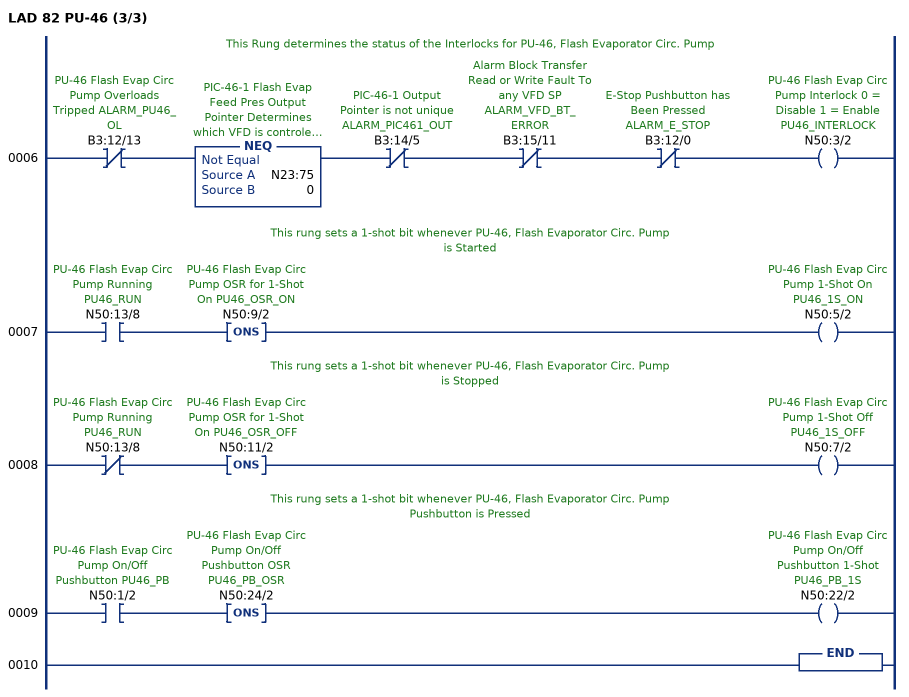
% Rung: 6 %
% This Rung determines the status of the Interlocks for PU-46, Flash Evaporator Circ. Pump %
SOR XIO B3:12/13 NEQ N23:75 0 XIO B3:14/5 XIO B3:15/11 XIO B3:12/0 OTE N50:3/2 EOR
%   B3:12/13  ALARM_PU46_OL  "PU-46 Flash Evap Circ Pump Overloads Tripped" %
%   N23:75  PIC461_OUT_PTR  "PIC-46-1 Flash Evap Feed Pres Output Pointer Determines which VFD is controled by FIC" %
%   B3:14/5  ALARM_PIC461_OUT  "PIC-46-1 Output Pointer is not unique" %
%   B3:15/11  ALARM_VFD_BT_ERROR  "Alarm Block Transfer Read or Write Fault To any VFD SP" %
%   B3:12/0  ALARM_E_STOP  "E-Stop Pushbutton has Been Pressed" %
%   N50:3/2  PU46_INTERLOCK  "PU-46 Flash Evap Circ Pump Interlock 0 = Disable 1 = Enable" %
% Rung: 7 %
% This rung sets a 1-shot bit whenever PU-46, Flash Evaporator Circ. Pump
% is Started %
SOR XIC N50:13/8 OSR N50:9/2 OTE N50:5/2 EOR
%   N50:13/8  PU46_RUN  "PU-46 Flash Evap Circ Pump Running" %
%   N50:9/2  PU46_OSR_ON  "PU-46 Flash Evap Circ Pump OSR for 1-Shot On" %
%   N50:5/2  PU46_1S_ON  "PU-46 Flash Evap Circ Pump 1-Shot On" %
% Rung: 8 %
% This rung sets a 1-shot bit whenever PU-46, Flash Evaporator Circ. Pump
% is Stopped %
SOR XIO N50:13/8 OSR N50:11/2 OTE N50:7/2 EOR
%   N50:13/8  PU46_RUN  "PU-46 Flash Evap Circ Pump Running" %
%   N50:11/2  PU46_OSR_OFF  "PU-46 Flash Evap Circ Pump OSR for 1-Shot On" %
%   N50:7/2  PU46_1S_OFF  "PU-46 Flash Evap Circ Pump 1-Shot Off" %
% Rung: 9 %
% This rung sets a 1-shot bit whenever PU-46, Flash Evaporator Circ. Pump
% Pushbutton is Pressed %
SOR XIC N50:1/2 OSR N50:24/2 OTE N50:22/2 EOR
%   N50:1/2  PU46_PB  "PU-46 Flash Evap Circ Pump On/Off Pushbutton" %
%   N50:24/2  PU46_PB_OSR  "PU-46 Flash Evap Circ Pump On/Off Pushbutton OSR" %
%   N50:22/2  PU46_PB_1S  "PU-46 Flash Evap Circ Pump On/Off Pushbutton 1-Shot" %
% Rung: 10 %
SOR END EOR

LADDER 86 "ALL VFDS"    % Control All VFD's %
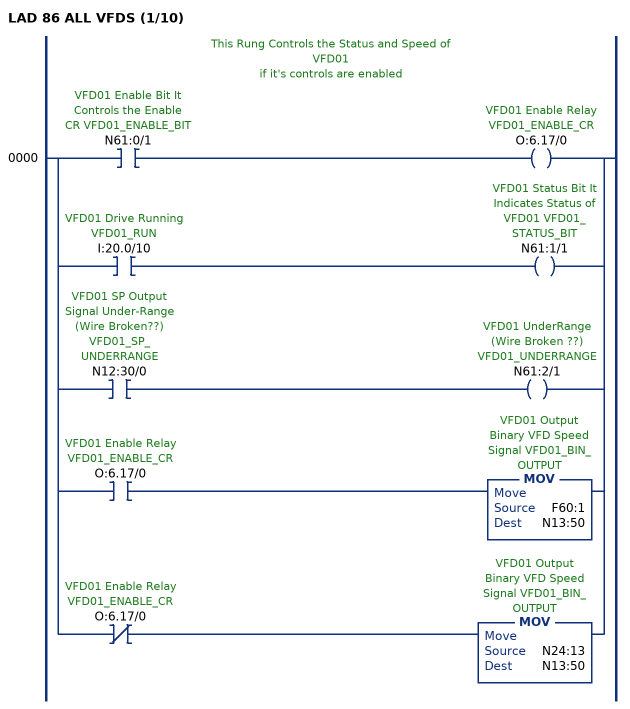
% Rung: 0 %
% This Rung Controls the Status and Speed of
% VFD01
% if it's controls are enabled %
SOR BST XIC N61:0/1 OTE O:6.17/0 NXB XIC I:20.0/10 OTE N61:1/1 NXB XIC N12:30/0 OTE N61:2/1 NXB XIC O:6.17/0 MOV F60:1 N13:50 NXB XIO O:6.17/0 MOV N24:13 N13:50 BND EOR
%   N61:0/1  VFD01_ENABLE_BIT  "VFD01 Enable Bit It Controls the Enable CR" %
%   O:6.17/0  VFD01_ENABLE_CR  "VFD01 Enable Relay" %
%   I:20.0/10  VFD01_RUN  "VFD01 Drive Running" %
%   N61:1/1  VFD01_STATUS_BIT  "VFD01 Status Bit It Indicates Status of VFD01" %
%   N12:30/0  VFD01_SP_UNDERRANGE  "VFD01 SP Output Signal Under-Range (Wire Broken??)" %
%   N61:2/1  VFD01_UNDERRANGE  "VFD01 UnderRange (Wire Broken ??)" %
%   F60:1  VFD01_BIN  "VFD01 VFD Table Value (is sent to Actual AO Location for VFD)" %
%   N13:50  VFD01_BIN_OUTPUT  "VFD01 Output Binary VFD Speed Signal" %
%   N24:13  AO_MIN_OE4  "Analog Output Minimum Value Generates 4 mA DC (To OE4 AO Module)" %

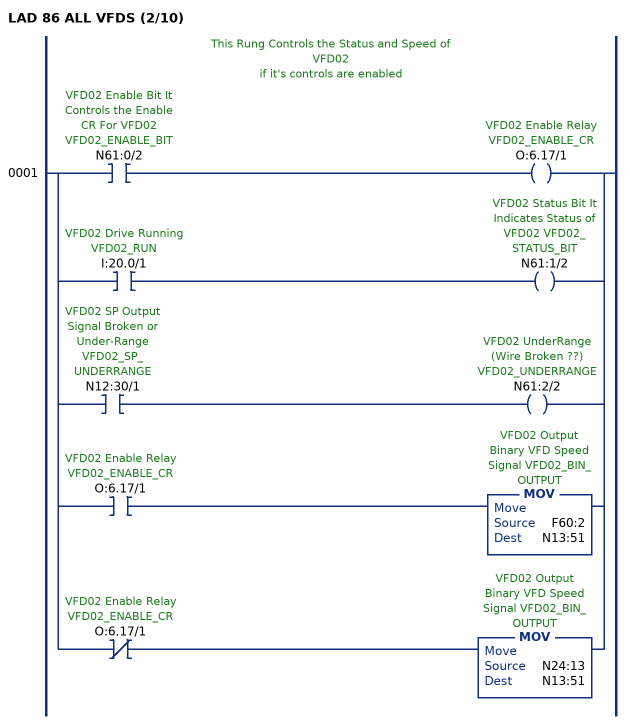
% Rung: 1 %
% This Rung Controls the Status and Speed of
% VFD02
% if it's controls are enabled %
SOR BST XIC N61:0/2 OTE O:6.17/1 NXB XIC I:20.0/1 OTE N61:1/2 NXB XIC N12:30/1 OTE N61:2/2 NXB XIC O:6.17/1 MOV F60:2 N13:51 NXB XIO O:6.17/1 MOV N24:13 N13:51 BND EOR
%   N61:0/2  VFD02_ENABLE_BIT  "VFD02 Enable Bit It Controls the Enable CR For VFD02" %
%   O:6.17/1  VFD02_ENABLE_CR  "VFD02 Enable Relay" %
%   I:20.0/1  VFD02_RUN  "VFD02 Drive Running" %
%   N61:1/2  VFD02_STATUS_BIT  "VFD02 Status Bit It Indicates Status of VFD02" %
%   N12:30/1  VFD02_SP_UNDERRANGE  "VFD02 SP Output Signal Broken or Under-Range" %
%   N61:2/2  VFD02_UNDERRANGE  "VFD02 UnderRange (Wire Broken ??)" %
%   F60:2  VFD02_BIN  "VFD02 VFD Table Value (is sent to Actual AO Location for VFD)" %
%   N13:51  VFD02_BIN_OUTPUT  "VFD02 Output Binary VFD Speed Signal" %
%   N24:13  AO_MIN_OE4  "Analog Output Minimum Value Generates 4 mA DC (To OE4 AO Module)" %

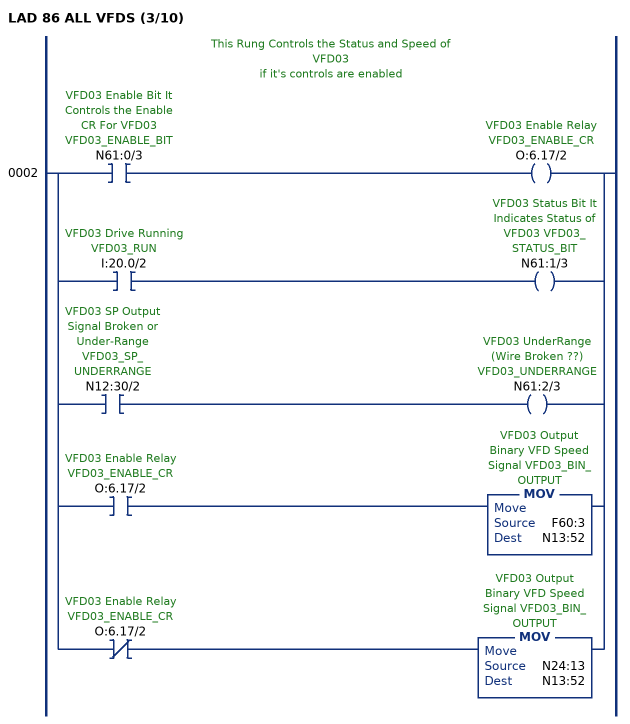
% Rung: 2 %
% This Rung Controls the Status and Speed of
% VFD03
% if it's controls are enabled %
SOR BST XIC N61:0/3 OTE O:6.17/2 NXB XIC I:20.0/2 OTE N61:1/3 NXB XIC N12:30/2 OTE N61:2/3 NXB XIC O:6.17/2 MOV F60:3 N13:52 NXB XIO O:6.17/2 MOV N24:13 N13:52 BND EOR
%   N61:0/3  VFD03_ENABLE_BIT  "VFD03 Enable Bit It Controls the Enable CR For VFD03" %
%   O:6.17/2  VFD03_ENABLE_CR  "VFD03 Enable Relay" %
%   I:20.0/2  VFD03_RUN  "VFD03 Drive Running" %
%   N61:1/3  VFD03_STATUS_BIT  "VFD03 Status Bit It Indicates Status of VFD03" %
%   N12:30/2  VFD03_SP_UNDERRANGE  "VFD03 SP Output Signal Broken or Under-Range" %
%   N61:2/3  VFD03_UNDERRANGE  "VFD03 UnderRange (Wire Broken ??)" %
%   F60:3  VFD03_BIN  "VFD03 VFD Table Value (is sent to Actual AO Location for VFD)" %
%   N13:52  VFD03_BIN_OUTPUT  "VFD03 Output Binary VFD Speed Signal" %
%   N24:13  AO_MIN_OE4  "Analog Output Minimum Value Generates 4 mA DC (To OE4 AO Module)" %

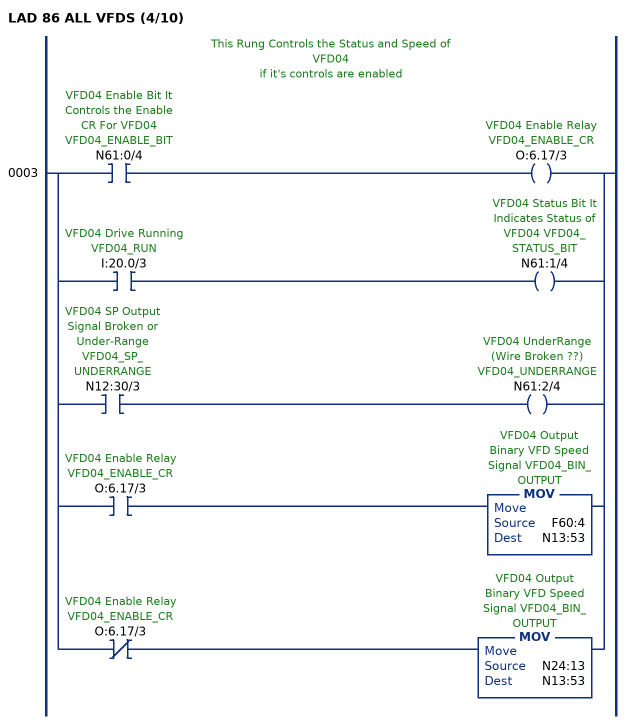
% Rung: 3 %
% This Rung Controls the Status and Speed of
% VFD04
% if it's controls are enabled %
SOR BST XIC N61:0/4 OTE O:6.17/3 NXB XIC I:20.0/3 OTE N61:1/4 NXB XIC N12:30/3 OTE N61:2/4 NXB XIC O:6.17/3 MOV F60:4 N13:53 NXB XIO O:6.17/3 MOV N24:13 N13:53 BND EOR
%   N61:0/4  VFD04_ENABLE_BIT  "VFD04 Enable Bit It Controls the Enable CR For VFD04" %
%   O:6.17/3  VFD04_ENABLE_CR  "VFD04 Enable Relay" %
%   I:20.0/3  VFD04_RUN  "VFD04 Drive Running" %
%   N61:1/4  VFD04_STATUS_BIT  "VFD04 Status Bit It Indicates Status of VFD04" %
%   N12:30/3  VFD04_SP_UNDERRANGE  "VFD04 SP Output Signal Broken or Under-Range" %
%   N61:2/4  VFD04_UNDERRANGE  "VFD04 UnderRange (Wire Broken ??)" %
%   F60:4  VFD04_BIN  "VFD04 VFD Table Value (is sent to Actual AO Location for VFD)" %
%   N13:53  VFD04_BIN_OUTPUT  "VFD04 Output Binary VFD Speed Signal" %
%   N24:13  AO_MIN_OE4  "Analog Output Minimum Value Generates 4 mA DC (To OE4 AO Module)" %

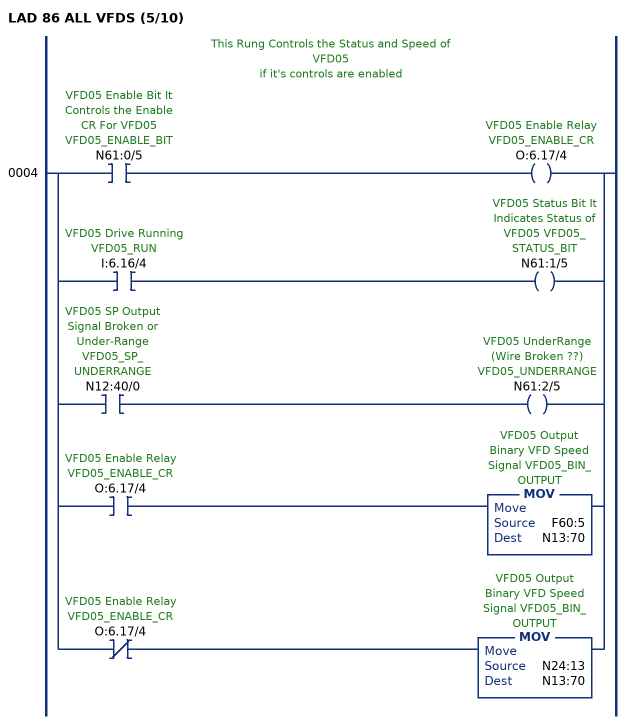
% Rung: 4 %
% This Rung Controls the Status and Speed of
% VFD05
% if it's controls are enabled %
SOR BST XIC N61:0/5 OTE O:6.17/4 NXB XIC I:6.16/4 OTE N61:1/5 NXB XIC N12:40/0 OTE N61:2/5 NXB XIC O:6.17/4 MOV F60:5 N13:70 NXB XIO O:6.17/4 MOV N24:13 N13:70 BND EOR
%   N61:0/5  VFD05_ENABLE_BIT  "VFD05 Enable Bit It Controls the Enable CR For VFD05" %
%   O:6.17/4  VFD05_ENABLE_CR  "VFD05 Enable Relay" %
%   I:6.16/4  VFD05_RUN  "VFD05 Drive Running" %
%   N61:1/5  VFD05_STATUS_BIT  "VFD05 Status Bit It Indicates Status of VFD05" %
%   N12:40/0  VFD05_SP_UNDERRANGE  "VFD05 SP Output Signal Broken or Under-Range" %
%   N61:2/5  VFD05_UNDERRANGE  "VFD05 UnderRange (Wire Broken ??)" %
%   F60:5  VFD05_BIN  "VFD05 VFD Table Value (is sent to Actual AO Location for VFD)" %
%   N13:70  VFD05_BIN_OUTPUT  "VFD05 Output Binary VFD Speed Signal" %
%   N24:13  AO_MIN_OE4  "Analog Output Minimum Value Generates 4 mA DC (To OE4 AO Module)" %

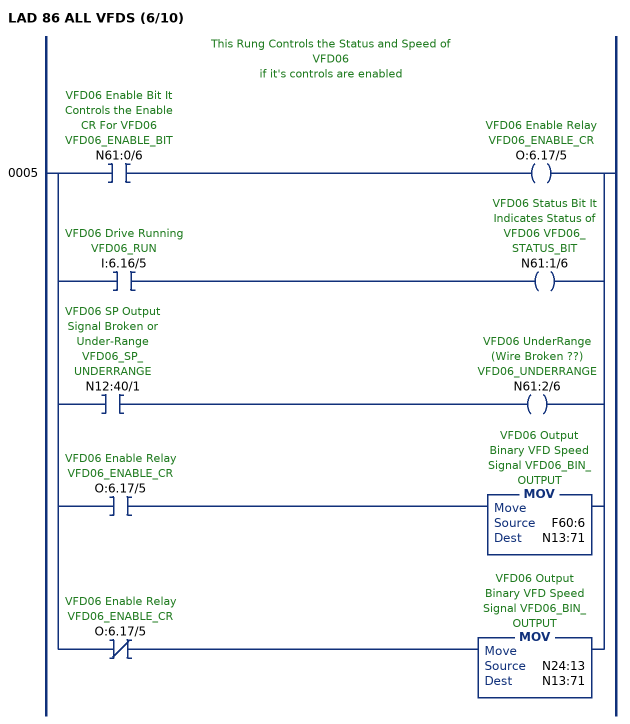
% Rung: 5 %
% This Rung Controls the Status and Speed of
% VFD06
% if it's controls are enabled %
SOR BST XIC N61:0/6 OTE O:6.17/5 NXB XIC I:6.16/5 OTE N61:1/6 NXB XIC N12:40/1 OTE N61:2/6 NXB XIC O:6.17/5 MOV F60:6 N13:71 NXB XIO O:6.17/5 MOV N24:13 N13:71 BND EOR
%   N61:0/6  VFD06_ENABLE_BIT  "VFD06 Enable Bit It Controls the Enable CR For VFD06" %
%   O:6.17/5  VFD06_ENABLE_CR  "VFD06 Enable Relay" %
%   I:6.16/5  VFD06_RUN  "VFD06 Drive Running" %
%   N61:1/6  VFD06_STATUS_BIT  "VFD06 Status Bit It Indicates Status of VFD06" %
%   N12:40/1  VFD06_SP_UNDERRANGE  "VFD06 SP Output Signal Broken or Under-Range" %
%   N61:2/6  VFD06_UNDERRANGE  "VFD06 UnderRange (Wire Broken ??)" %
%   F60:6  VFD06_BIN  "VFD06 VFD Table Value (is sent to Actual AO Location for VFD)" %
%   N13:71  VFD06_BIN_OUTPUT  "VFD06 Output Binary VFD Speed Signal" %
%   N24:13  AO_MIN_OE4  "Analog Output Minimum Value Generates 4 mA DC (To OE4 AO Module)" %

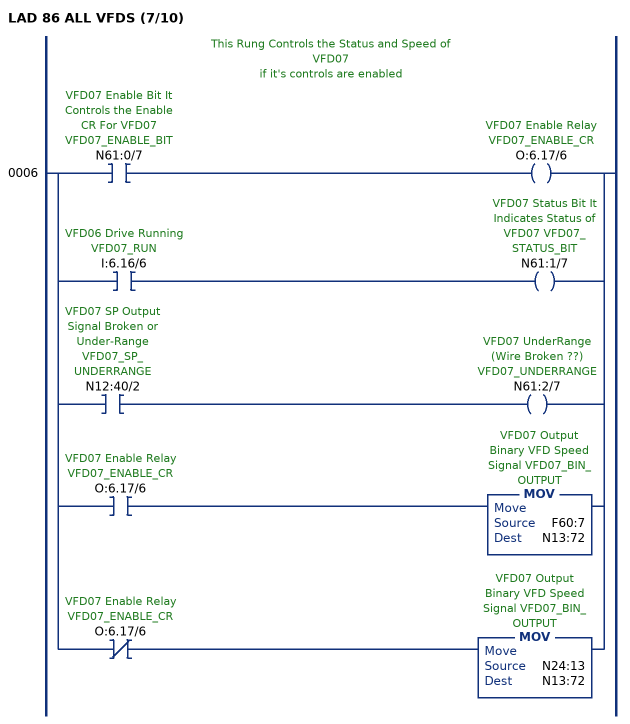
% Rung: 6 %
% This Rung Controls the Status and Speed of
% VFD07
% if it's controls are enabled %
SOR BST XIC N61:0/7 OTE O:6.17/6 NXB XIC I:6.16/6 OTE N61:1/7 NXB XIC N12:40/2 OTE N61:2/7 NXB XIC O:6.17/6 MOV F60:7 N13:72 NXB XIO O:6.17/6 MOV N24:13 N13:72 BND EOR
%   N61:0/7  VFD07_ENABLE_BIT  "VFD07 Enable Bit It Controls the Enable CR For VFD07" %
%   O:6.17/6  VFD07_ENABLE_CR  "VFD07 Enable Relay" %
%   I:6.16/6  VFD07_RUN  "VFD06 Drive Running" %
%   N61:1/7  VFD07_STATUS_BIT  "VFD07 Status Bit It Indicates Status of VFD07" %
%   N12:40/2  VFD07_SP_UNDERRANGE  "VFD07 SP Output Signal Broken or Under-Range" %
%   N61:2/7  VFD07_UNDERRANGE  "VFD07 UnderRange (Wire Broken ??)" %
%   F60:7  VFD07_BIN  "VFD07 VFD Table Value (is sent to Actual AO Location for VFD)" %
%   N13:72  VFD07_BIN_OUTPUT  "VFD07 Output Binary VFD Speed Signal" %
%   N24:13  AO_MIN_OE4  "Analog Output Minimum Value Generates 4 mA DC (To OE4 AO Module)" %

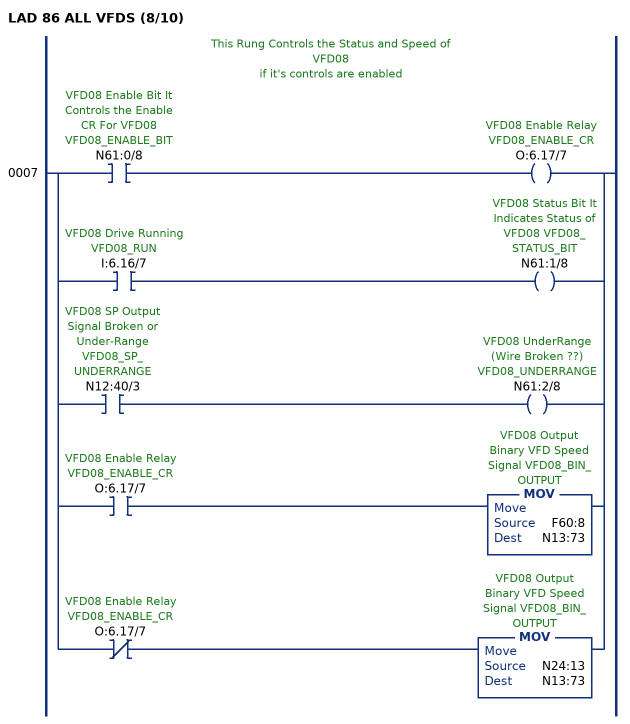
% Rung: 7 %
% This Rung Controls the Status and Speed of
% VFD08
% if it's controls are enabled %
SOR BST XIC N61:0/8 OTE O:6.17/7 NXB XIC I:6.16/7 OTE N61:1/8 NXB XIC N12:40/3 OTE N61:2/8 NXB XIC O:6.17/7 MOV F60:8 N13:73 NXB XIO O:6.17/7 MOV N24:13 N13:73 BND EOR
%   N61:0/8  VFD08_ENABLE_BIT  "VFD08 Enable Bit It Controls the Enable CR For VFD08" %
%   O:6.17/7  VFD08_ENABLE_CR  "VFD08 Enable Relay" %
%   I:6.16/7  VFD08_RUN  "VFD08 Drive Running" %
%   N61:1/8  VFD08_STATUS_BIT  "VFD08 Status Bit It Indicates Status of VFD08" %
%   N12:40/3  VFD08_SP_UNDERRANGE  "VFD08 SP Output Signal Broken or Under-Range" %
%   N61:2/8  VFD08_UNDERRANGE  "VFD08 UnderRange (Wire Broken ??)" %
%   F60:8  VFD08_BIN  "VFD08 VFD Table Value (is sent to Actual AO Location for VFD)" %
%   N13:73  VFD08_BIN_OUTPUT  "VFD08 Output Binary VFD Speed Signal" %
%   N24:13  AO_MIN_OE4  "Analog Output Minimum Value Generates 4 mA DC (To OE4 AO Module)" %

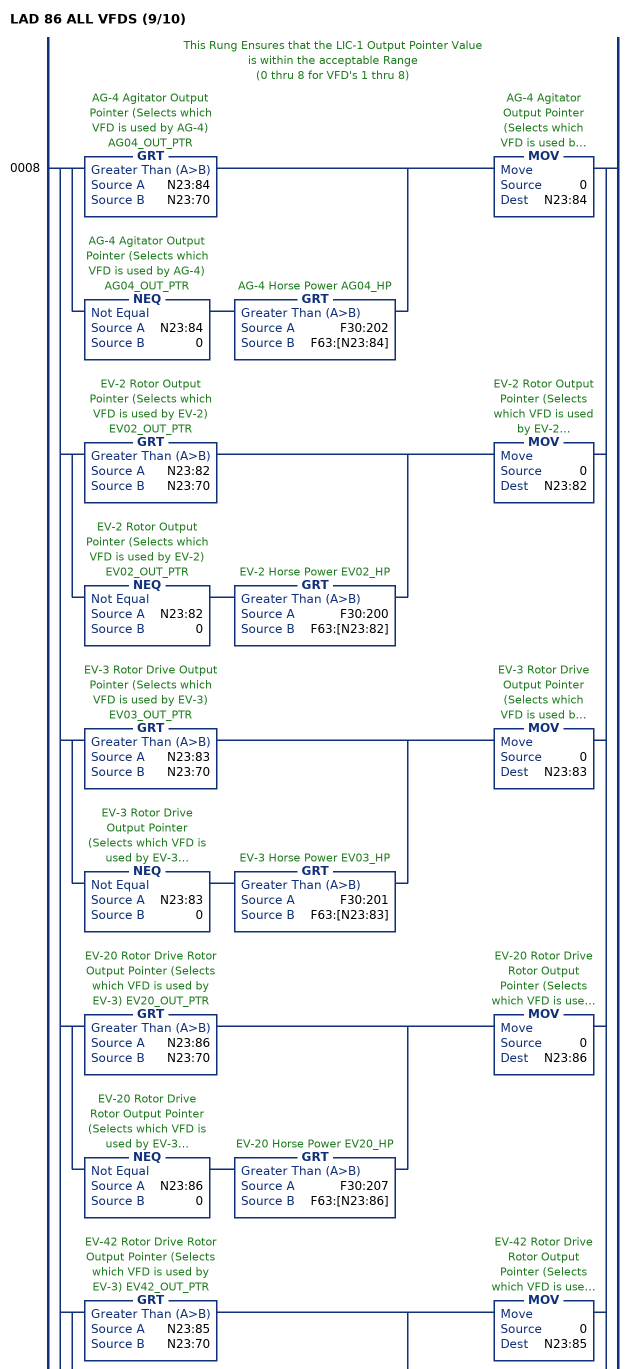

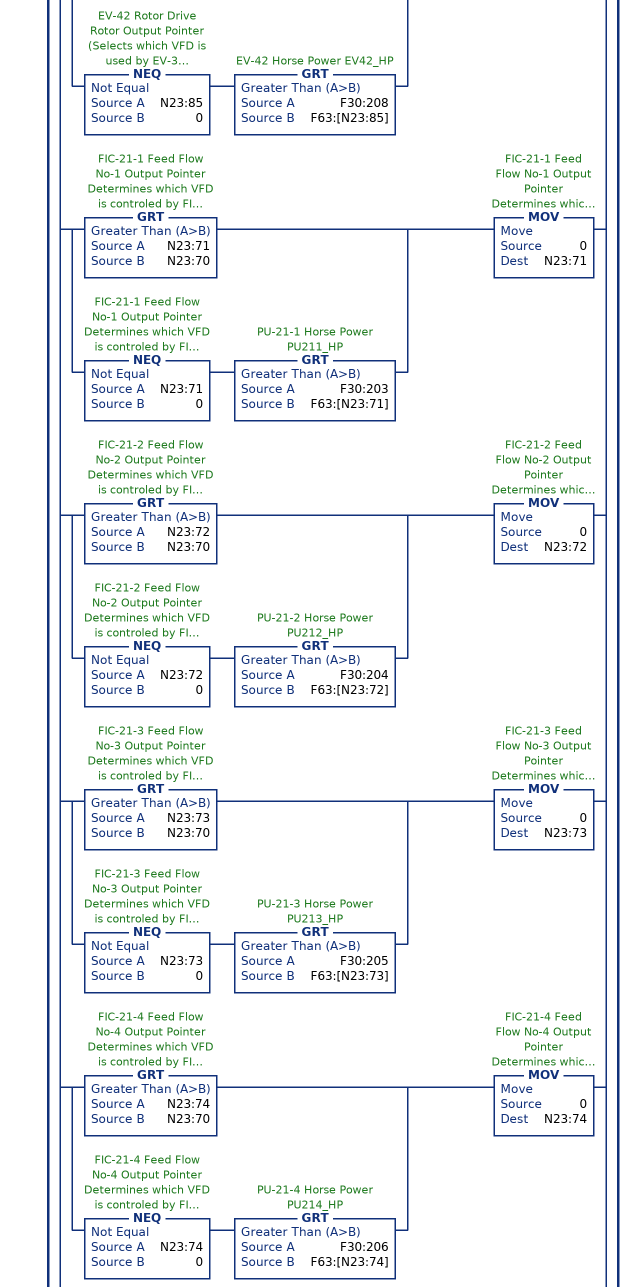

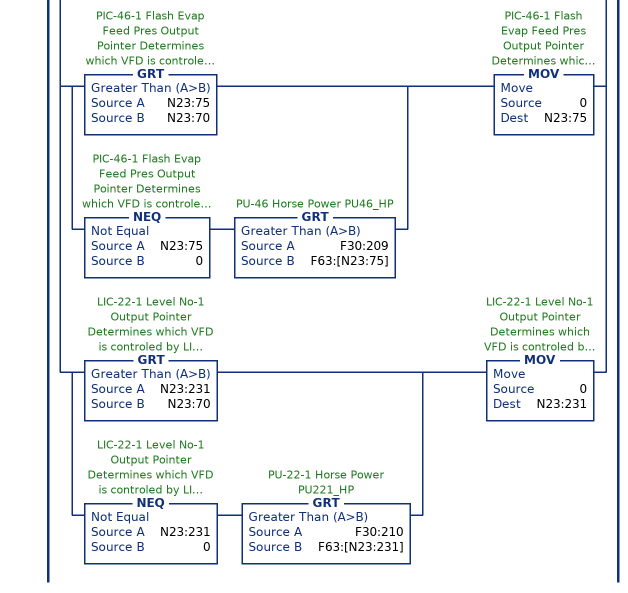
% Rung: 8 %
% This Rung Ensures that the LIC-1 Output Pointer Value
% is within the acceptable Range
% (0 thru 8 for VFD's 1 thru 8) %
SOR BST BST GRT N23:84 N23:70 NXB NEQ N23:84 0 GRT F30:202 F63:[N23:84] BND MOV 0 N23:84 NXB BST GRT N23:82 N23:70 NXB NEQ N23:82 0 GRT F30:200 F63:[N23:82] BND MOV 0 N23:82 NXB BST GRT N23:83 N23:70 NXB NEQ N23:83 0 GRT F30:201 F63:[N23:83] BND MOV 0 N23:83 NXB BST GRT N23:86 N23:70 NXB NEQ N23:86 0 GRT F30:207 F63:[N23:86] BND MOV 0 N23:86 NXB BST GRT N23:85 N23:70 NXB NEQ N23:85 0 GRT F30:208 F63:[N23:85] BND MOV 0 N23:85 NXB BST GRT N23:71 N23:70 NXB NEQ N23:71 0 GRT F30:203 F63:[N23:71] BND MOV 0 N23:71 NXB BST GRT N23:72 N23:70 NXB NEQ N23:72 0 GRT F30:204 F63:[N23:72] BND MOV 0 N23:72 NXB BST GRT N23:73 N23:70 NXB NEQ N23:73 0 GRT F30:205 F63:[N23:73] BND MOV 0 N23:73 NXB BST GRT N23:74 N23:70 NXB NEQ N23:74 0 GRT F30:206 F63:[N23:74] BND MOV 0 N23:74 NXB BST GRT N23:75 N23:70 NXB NEQ N23:75 0 GRT F30:209 F63:[N23:75] BND MOV 0 N23:75 NXB BST GRT N23:231 N23:70 NXB NEQ N23:231 0 GRT F30:210 F63:[N23:231] BND MOV 0 N23:231 BND EOR
%   N23:84  AG04_OUT_PTR  "AG-4 Agitator Output Pointer (Selects which VFD is used by AG-4)" %
%   N23:70  MAX_VFD_ALLOWED  "Maximum Number of VFDs Available" %
%   F30:202  AG04_HP  "AG-4 Horse Power" %
%   N23:82  EV02_OUT_PTR  "EV-2 Rotor Output Pointer (Selects which VFD is used by EV-2)" %
%   F30:200  EV02_HP  "EV-2 Horse Power" %
%   N23:83  EV03_OUT_PTR  "EV-3 Rotor Drive Output Pointer (Selects which VFD is used by EV-3)" %
%   F30:201  EV03_HP  "EV-3 Horse Power" %
%   N23:86  EV20_OUT_PTR  "EV-20 Rotor Drive Rotor Output Pointer (Selects which VFD is used by EV-3)" %
%   F30:207  EV20_HP  "EV-20 Horse Power" %
%   N23:85  EV42_OUT_PTR  "EV-42 Rotor Drive Rotor Output Pointer (Selects which VFD is used by EV-3)" %
%   F30:208  EV42_HP  "EV-42 Horse Power" %
%   N23:71  FIC211_OUT_PTR  "FIC-21-1 Feed Flow No-1 Output Pointer Determines which VFD is controled by FIC" %
%   F30:203  PU211_HP  "PU-21-1 Horse Power" %
%   N23:72  FIC212_OUT_PTR  "FIC-21-2 Feed Flow No-2 Output Pointer Determines which VFD is controled by FIC" %
%   F30:204  PU212_HP  "PU-21-2 Horse Power" %
%   N23:73  FIC213_OUT_PTR  "FIC-21-3 Feed Flow No-3 Output Pointer Determines which VFD is controled by FIC" %
%   F30:205  PU213_HP  "PU-21-3 Horse Power" %
%   N23:74  FIC214_OUT_PTR  "FIC-21-4 Feed Flow No-4 Output Pointer Determines which VFD is controled by FIC" %
%   F30:206  PU214_HP  "PU-21-4 Horse Power" %
%   N23:75  PIC461_OUT_PTR  "PIC-46-1 Flash Evap Feed Pres Output Pointer Determines which VFD is controled by FIC" %
%   F30:209  PU46_HP  "PU-46 Horse Power" %
%   N23:231  LIC221_OUT_PTR  "LIC-22-1 Level No-1 Output Pointer Determines which VFD is controled by LIC" %
%   F30:210  PU221_HP  "PU-22-1 Horse Power" %

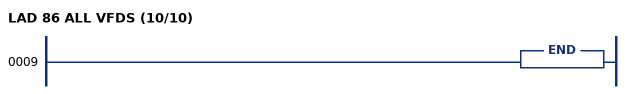
% Rung: 9 %
SOR END EOR

LADDER 90 "ALL PIDS"    % Execute All PID Statements using STI Interupt %
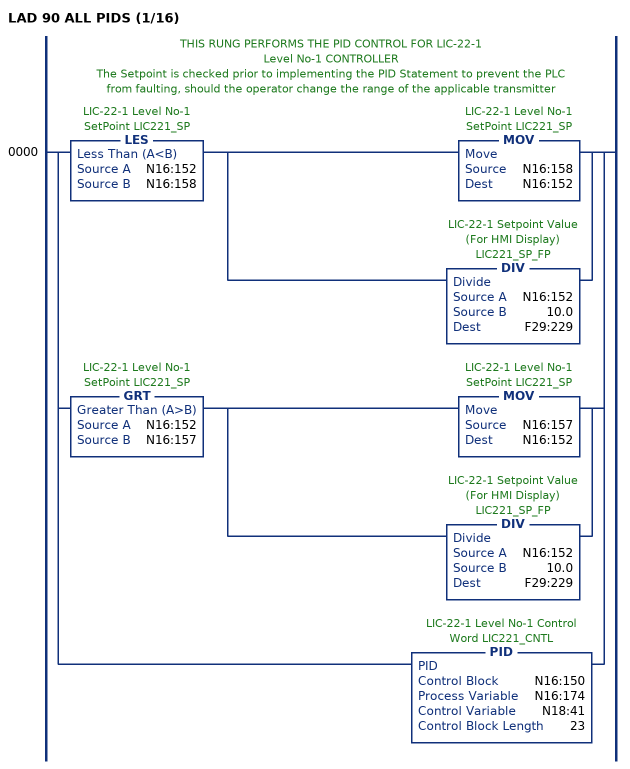
% Rung: 0 %
% THIS RUNG PERFORMS THE PID CONTROL FOR LIC-22-1
% Level No-1 CONTROLLER
% The Setpoint is checked prior to implementing the PID Statement to prevent the PLC
% from faulting, should the operator change the range of the applicable transmitter %
SOR BST LES N16:152 N16:158 BST MOV N16:158 N16:152 NXB DIV N16:152 10.0 F29:229 BND NXB GRT N16:152 N16:157 BST MOV N16:157 N16:152 NXB DIV N16:152 10.0 F29:229 BND NXB PID N16:150 N16:174 N18:41 23 BND EOR
%   N16:152  LIC221_SP  "LIC-22-1 Level No-1 SetPoint" %
%   N16:158  LIC221_SMIN  "LIC-22-1 Level No-1 Setpoint Minimum" %
%   F29:229  LIC221_SP_FP  "LIC-22-1 Setpoint Value (For HMI Display)" %
%   N16:157  LIC221_SMAX  "LIC-22-1 Level No-1 Setpoint Maximum" %
%   N16:150  LIC221_CNTL  "LIC-22-1 Level No-1 Control Word" %
%   N16:174  LIC221_IN  "LIC-22-1 Level No-1 Scaled Input" %
%   N18:41  LIC221_OUT1  "LIC-22-1 Level No-1 PID Output Value" %

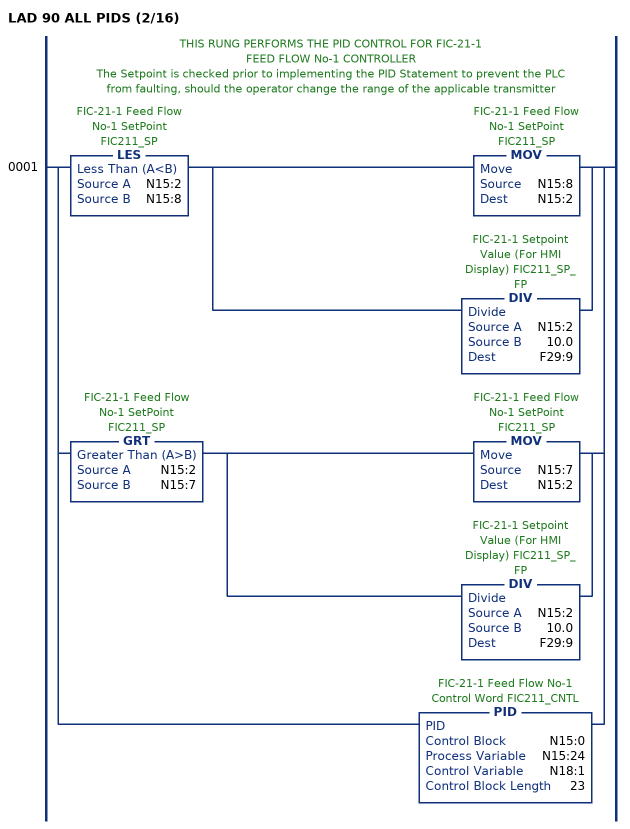
% Rung: 1 %
% THIS RUNG PERFORMS THE PID CONTROL FOR FIC-21-1
% FEED FLOW No-1 CONTROLLER
% The Setpoint is checked prior to implementing the PID Statement to prevent the PLC
% from faulting, should the operator change the range of the applicable transmitter %
SOR BST LES N15:2 N15:8 BST MOV N15:8 N15:2 NXB DIV N15:2 10.0 F29:9 BND NXB GRT N15:2 N15:7 BST MOV N15:7 N15:2 NXB DIV N15:2 10.0 F29:9 BND NXB PID N15:0 N15:24 N18:1 23 BND EOR
%   N15:2  FIC211_SP  "FIC-21-1 Feed Flow No-1 SetPoint" %
%   N15:8  FIC211_SMIN  "FIC-21-1 Feed Flow No-1 Setpoint Minimum" %
%   F29:9  FIC211_SP_FP  "FIC-21-1 Setpoint Value (For HMI Display)" %
%   N15:7  FIC211_SMAX  "FIC-21-1 Feed Flow No-1 Setpoint Maximum" %
%   N15:0  FIC211_CNTL  "FIC-21-1 Feed Flow No-1 Control Word" %
%   N15:24  FIC211_IN  "FIC-21-1 Feed Flow No-1 Scaled Input" %
%   N18:1  FIC211_OUT1  "FIC-21-1 Feed Flow No-1 PID Output Value" %

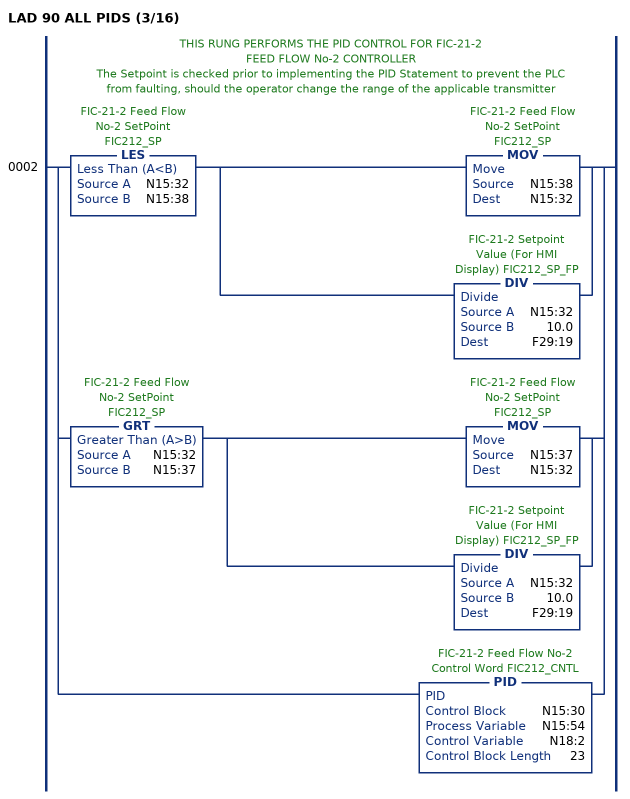
% Rung: 2 %
% THIS RUNG PERFORMS THE PID CONTROL FOR FIC-21-2
% FEED FLOW No-2 CONTROLLER
%  The Setpoint is checked prior to implementing the PID Statement to prevent the PLC
% from faulting, should the operator change the range of the applicable transmitter %
SOR BST LES N15:32 N15:38 BST MOV N15:38 N15:32 NXB DIV N15:32 10.0 F29:19 BND NXB GRT N15:32 N15:37 BST MOV N15:37 N15:32 NXB DIV N15:32 10.0 F29:19 BND NXB PID N15:30 N15:54 N18:2 23 BND EOR
%   N15:32  FIC212_SP  "FIC-21-2 Feed Flow No-2 SetPoint" %
%   N15:38  FIC212_SMIN  "FIC-21-2 Feed Flow No-2 Setpoint Minimum" %
%   F29:19  FIC212_SP_FP  "FIC-21-2 Setpoint Value (For HMI Display)" %
%   N15:37  FIC212_SMAX  "FIC-21-2 Feed Flow No-2 Setpoint Maximum" %
%   N15:30  FIC212_CNTL  "FIC-21-2 Feed Flow No-2 Control Word" %
%   N15:54  FIC212_IN  "FIC-21-2 Feed Flow No-2 Scaled Input" %
%   N18:2  FIC212_OUT1  "FIC-21-2 Feed Flow No-2 PID Output Value" %

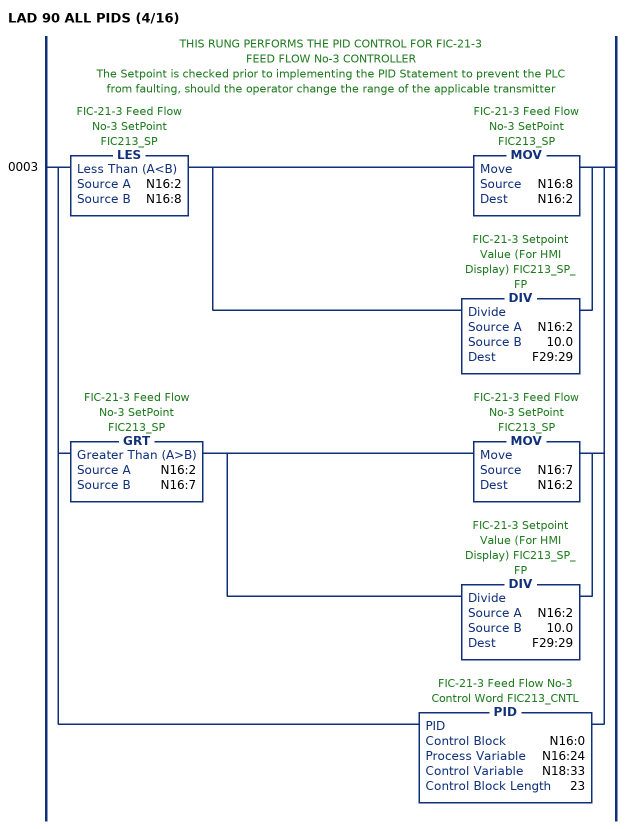
% Rung: 3 %
% THIS RUNG PERFORMS THE PID CONTROL FOR FIC-21-3
% FEED FLOW No-3 CONTROLLER
%  The Setpoint is checked prior to implementing the PID Statement to prevent the PLC
% from faulting, should the operator change the range of the applicable transmitter %
SOR BST LES N16:2 N16:8 BST MOV N16:8 N16:2 NXB DIV N16:2 10.0 F29:29 BND NXB GRT N16:2 N16:7 BST MOV N16:7 N16:2 NXB DIV N16:2 10.0 F29:29 BND NXB PID N16:0 N16:24 N18:33 23 BND EOR
%   N16:2  FIC213_SP  "FIC-21-3 Feed Flow No-3 SetPoint" %
%   N16:8  FIC213_SMIN  "FIC-21-3 Feed Flow No-3 Setpoint Minimum" %
%   F29:29  FIC213_SP_FP  "FIC-21-3 Setpoint Value (For HMI Display)" %
%   N16:7  FIC213_SMAX  "FIC-21-3 Feed Flow No-3 Setpoint Maximum" %
%   N16:0  FIC213_CNTL  "FIC-21-3 Feed Flow No-3 Control Word" %
%   N16:24  FIC213_IN  "FIC-21-3 Feed Flow No-3 Scaled Input" %
%   N18:33  FIC213_OUT1  "FIC-21-3 Feed Flow No-3 PID Output Value" %

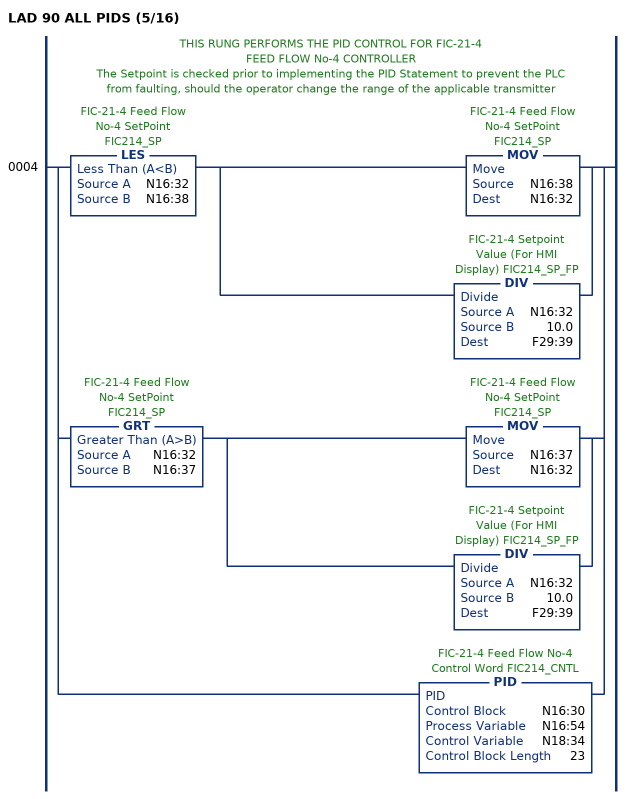
% Rung: 4 %
% THIS RUNG PERFORMS THE PID CONTROL FOR FIC-21-4
% FEED FLOW No-4 CONTROLLER
%  The Setpoint is checked prior to implementing the PID Statement to prevent the PLC
% from faulting, should the operator change the range of the applicable transmitter %
SOR BST LES N16:32 N16:38 BST MOV N16:38 N16:32 NXB DIV N16:32 10.0 F29:39 BND NXB GRT N16:32 N16:37 BST MOV N16:37 N16:32 NXB DIV N16:32 10.0 F29:39 BND NXB PID N16:30 N16:54 N18:34 23 BND EOR
%   N16:32  FIC214_SP  "FIC-21-4 Feed Flow No-4 SetPoint" %
%   N16:38  FIC214_SMIN  "FIC-21-4 Feed Flow No-4 Setpoint Minimum" %
%   F29:39  FIC214_SP_FP  "FIC-21-4 Setpoint Value (For HMI Display)" %
%   N16:37  FIC214_SMAX  "FIC-21-4 Feed Flow No-4 Setpoint Maximum" %
%   N16:30  FIC214_CNTL  "FIC-21-4 Feed Flow No-4 Control Word" %
%   N16:54  FIC214_IN  "FIC-21-4 Feed Flow No-4 Scaled Input" %
%   N18:34  FIC214_OUT1  "FIC-21-4 Feed Flow No-4 PID Output Value" %

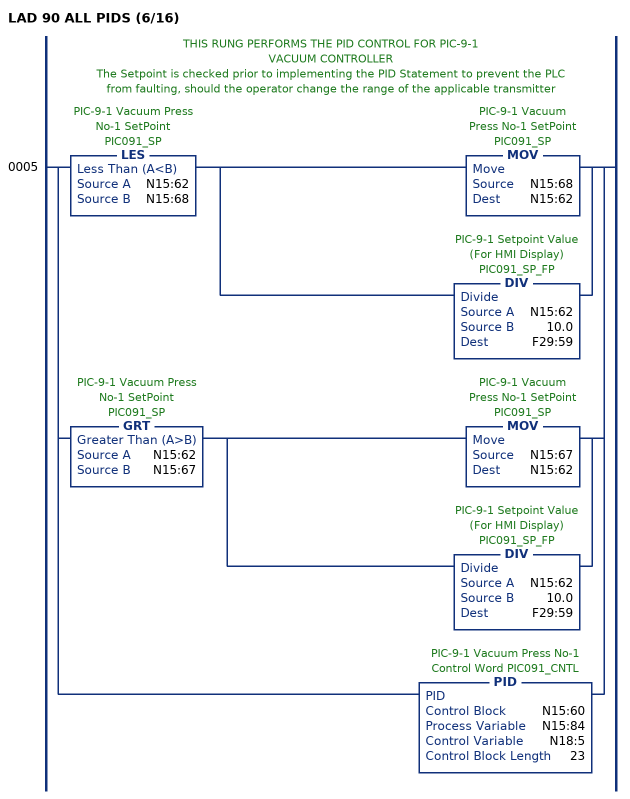
% Rung: 5 %
% THIS RUNG PERFORMS THE PID CONTROL FOR PIC-9-1
% VACUUM CONTROLLER
% The Setpoint is checked prior to implementing the PID Statement to prevent the PLC
% from faulting, should the operator change the range of the applicable transmitter %
SOR BST LES N15:62 N15:68 BST MOV N15:68 N15:62 NXB DIV N15:62 10.0 F29:59 BND NXB GRT N15:62 N15:67 BST MOV N15:67 N15:62 NXB DIV N15:62 10.0 F29:59 BND NXB PID N15:60 N15:84 N18:5 23 BND EOR
%   N15:62  PIC091_SP  "PIC-9-1 Vacuum Press No-1 SetPoint" %
%   N15:68  PIC091_SMIN  "PIC-9-1 Vacuum Press No-1 Setpoint Minimum" %
%   F29:59  PIC091_SP_FP  "PIC-9-1 Setpoint Value (For HMI Display)" %
%   N15:67  PIC091_SMAX  "PIC-9-1 Vacuum Press No-1 Setpoint Maximum" %
%   N15:60  PIC091_CNTL  "PIC-9-1 Vacuum Press No-1 Control Word" %
%   N15:84  PIC091_IN  "PIC-9-1 Vacuum Press No-1 Scaled Input" %
%   N18:5  PIC091_OUT1  "PIC-9-1 Vacuum Press No-1 PID Output Value" %

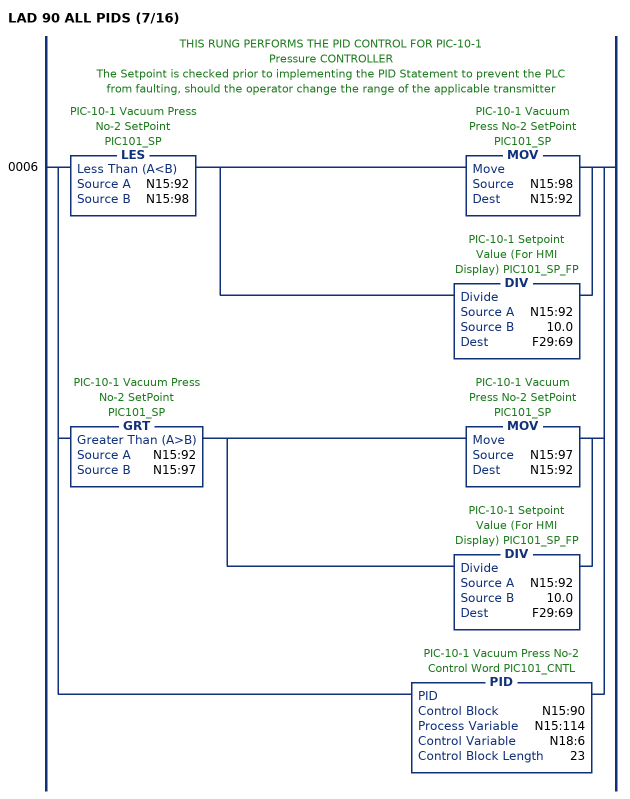
% Rung: 6 %
% THIS RUNG PERFORMS THE PID CONTROL FOR PIC-10-1
% Pressure CONTROLLER
% The Setpoint is checked prior to implementing the PID Statement to prevent the PLC
% from faulting, should the operator change the range of the applicable transmitter %
SOR BST LES N15:92 N15:98 BST MOV N15:98 N15:92 NXB DIV N15:92 10.0 F29:69 BND NXB GRT N15:92 N15:97 BST MOV N15:97 N15:92 NXB DIV N15:92 10.0 F29:69 BND NXB PID N15:90 N15:114 N18:6 23 BND EOR
%   N15:92  PIC101_SP  "PIC-10-1 Vacuum Press No-2 SetPoint" %
%   N15:98  PIC101_SMIN  "PIC-10-1 Vacuum Press No-2 Setpoint Minimum" %
%   F29:69  PIC101_SP_FP  "PIC-10-1 Setpoint Value (For HMI Display)" %
%   N15:97  PIC101_SMAX  "PIC-10-1 Vacuum Press No-2 Setpoint Maximum" %
%   N15:90  PIC101_CNTL  "PIC-10-1 Vacuum Press No-2 Control Word" %
%   N15:114  PIC101_IN  "PIC-10-1 Vacuum Press No-2 Scaled Input" %
%   N18:6  PIC101_OUT1  "PIC-10-1 Vacuum Press No-2 PID Output Value" %

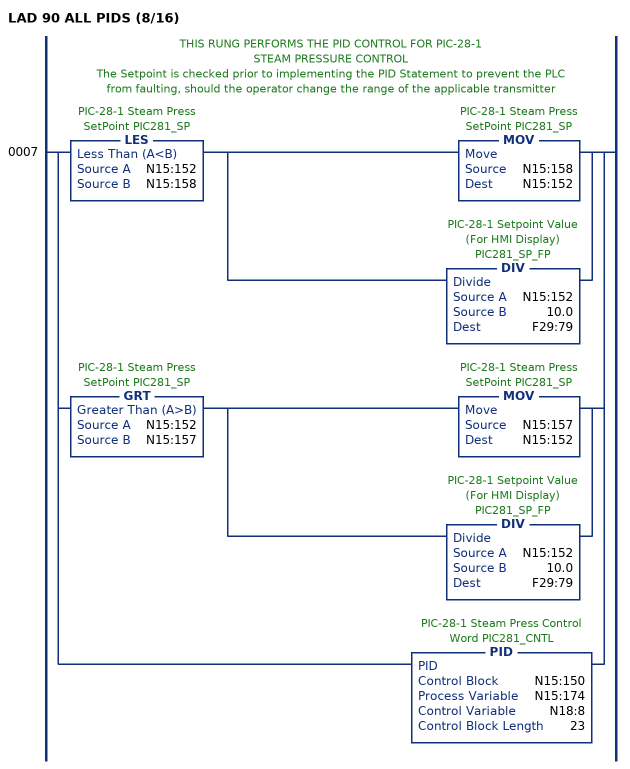
% Rung: 7 %
% THIS RUNG PERFORMS THE PID CONTROL FOR PIC-28-1
% STEAM PRESSURE CONTROL
% The Setpoint is checked prior to implementing the PID Statement to prevent the PLC
% from faulting, should the operator change the range of the applicable transmitter %
SOR BST LES N15:152 N15:158 BST MOV N15:158 N15:152 NXB DIV N15:152 10.0 F29:79 BND NXB GRT N15:152 N15:157 BST MOV N15:157 N15:152 NXB DIV N15:152 10.0 F29:79 BND NXB PID N15:150 N15:174 N18:8 23 BND EOR
%   N15:152  PIC281_SP  "PIC-28-1 Steam Press SetPoint" %
%   N15:158  PIC281_SMIN  "PIC-28-1 Steam Press Setpoint Minimum" %
%   F29:79  PIC281_SP_FP  "PIC-28-1 Setpoint Value (For HMI Display)" %
%   N15:157  PIC281_SMAX  "PIC-28-1 Steam Press Setpoint Maximum" %
%   N15:150  PIC281_CNTL  "PIC-28-1 Steam Press Control Word" %
%   N15:174  PIC281_IN  "PIC-28-1 Steam Press Scaled Input" %
%   N18:8  PIC281_OUT1  "PIC-28-1 Steam Press PID Output Value" %

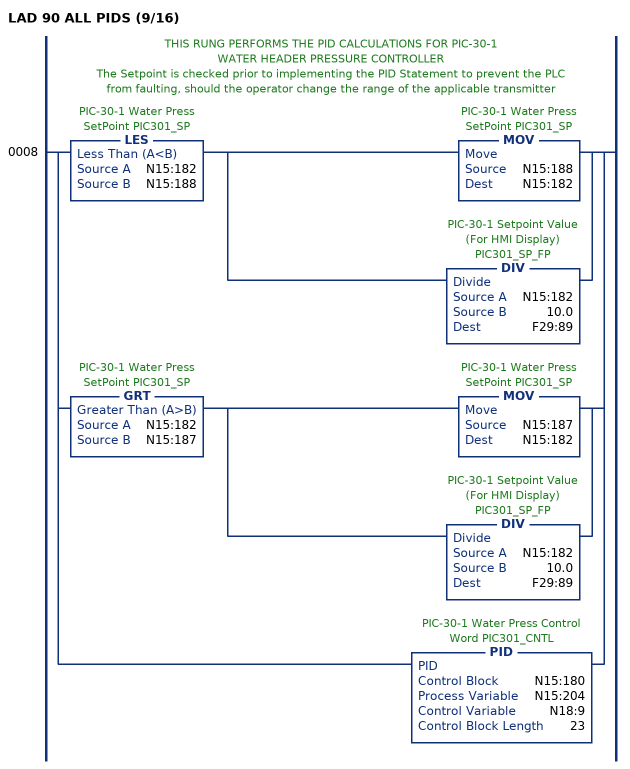
% Rung: 8 %
% THIS RUNG PERFORMS THE PID CALCULATIONS FOR PIC-30-1
% WATER HEADER PRESSURE CONTROLLER
% The Setpoint is checked prior to implementing the PID Statement to prevent the PLC
% from faulting, should the operator change the range of the applicable transmitter %
SOR BST LES N15:182 N15:188 BST MOV N15:188 N15:182 NXB DIV N15:182 10.0 F29:89 BND NXB GRT N15:182 N15:187 BST MOV N15:187 N15:182 NXB DIV N15:182 10.0 F29:89 BND NXB PID N15:180 N15:204 N18:9 23 BND EOR
%   N15:182  PIC301_SP  "PIC-30-1 Water Press SetPoint" %
%   N15:188  PIC301_SMIN  "PIC-30-1 Water Press Setpoint Minimum" %
%   F29:89  PIC301_SP_FP  "PIC-30-1 Setpoint Value (For HMI Display)" %
%   N15:187  PIC301_SMAX  "PIC-30-1 Water Press Setpoint Maximum" %
%   N15:180  PIC301_CNTL  "PIC-30-1 Water Press Control Word" %
%   N15:204  PIC301_IN  "PIC-30-1 Water Press Scaled Input" %
%   N18:9  PIC301_OUT1  "PIC-30-1 Water Press PID Output Value" %

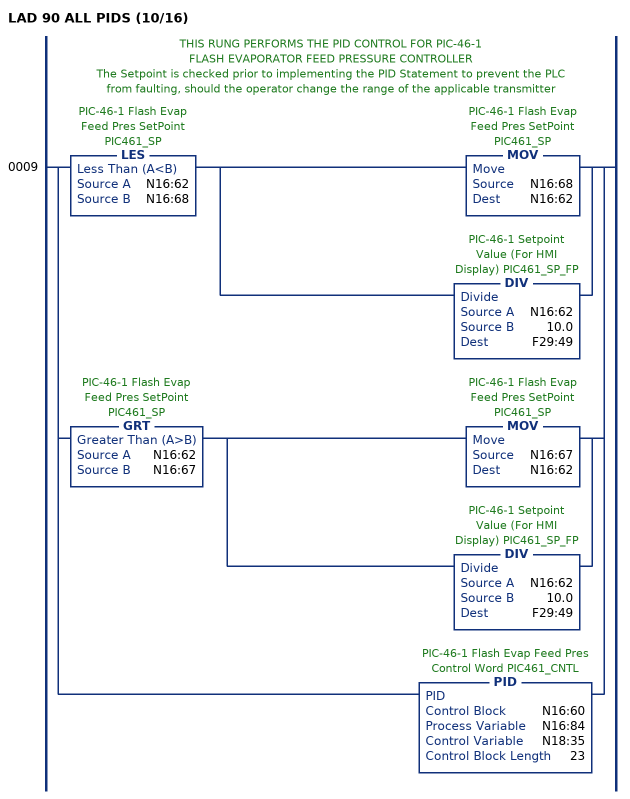
% Rung: 9 %
% THIS RUNG PERFORMS THE PID CONTROL FOR PIC-46-1
% FLASH EVAPORATOR FEED PRESSURE CONTROLLER
%  The Setpoint is checked prior to implementing the PID Statement to prevent the PLC
% from faulting, should the operator change the range of the applicable transmitter %
SOR BST LES N16:62 N16:68 BST MOV N16:68 N16:62 NXB DIV N16:62 10.0 F29:49 BND NXB GRT N16:62 N16:67 BST MOV N16:67 N16:62 NXB DIV N16:62 10.0 F29:49 BND NXB PID N16:60 N16:84 N18:35 23 BND EOR
%   N16:62  PIC461_SP  "PIC-46-1 Flash Evap Feed Pres SetPoint" %
%   N16:68  PIC461_SMIN  "PIC-46-1 Flash Evap Feed Pres Setpoint Minimum" %
%   F29:49  PIC461_SP_FP  "PIC-46-1 Setpoint Value (For HMI Display)" %
%   N16:67  PIC461_SMAX  "PIC-46-1 Flash Evap Feed Pres Setpoint Maximum" %
%   N16:60  PIC461_CNTL  "PIC-46-1 Flash Evap Feed Pres Control Word" %
%   N16:84  PIC461_IN  "PIC-46-1 Flash Evap Feed Pres Scaled Input" %
%   N18:35  PIC461_OUT1  "PIC-46-1 Flash Evap Feed Pres PID Output Value" %

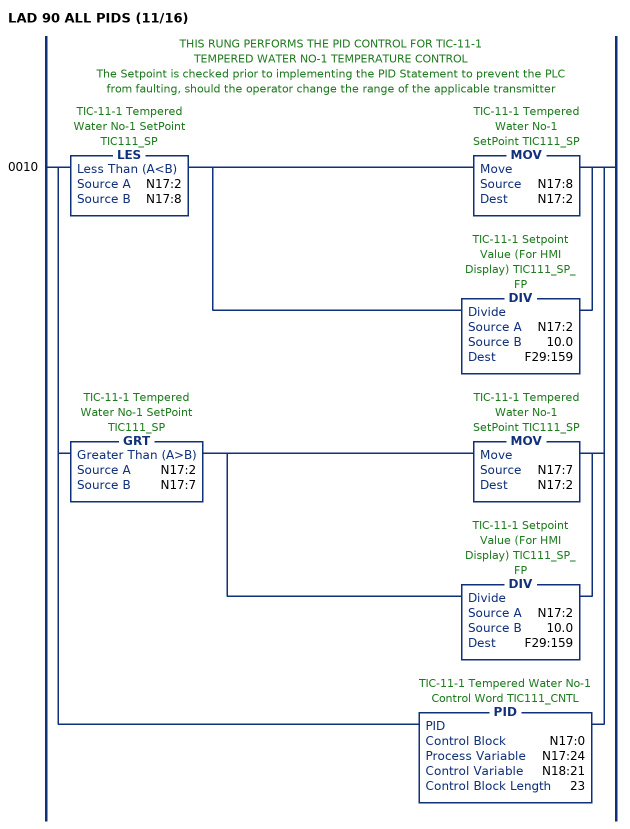
% Rung: 10 %
% THIS RUNG PERFORMS THE PID CONTROL FOR TIC-11-1
% TEMPERED WATER NO-1 TEMPERATURE CONTROL
% The Setpoint is checked prior to implementing the PID Statement to prevent the PLC
% from faulting, should the operator change the range of the applicable transmitter %
SOR BST LES N17:2 N17:8 BST MOV N17:8 N17:2 NXB DIV N17:2 10.0 F29:159 BND NXB GRT N17:2 N17:7 BST MOV N17:7 N17:2 NXB DIV N17:2 10.0 F29:159 BND NXB PID N17:0 N17:24 N18:21 23 BND EOR
%   N17:2  TIC111_SP  "TIC-11-1 Tempered Water No-1 SetPoint" %
%   N17:8  TIC111_SMIN  "TIC-11-1 Tempered Water No-1 Setpoint Minimum" %
%   F29:159  TIC111_SP_FP  "TIC-11-1 Setpoint Value (For HMI Display)" %
%   N17:7  TIC111_SMAX  "TIC-11-1 Tempered Water No-1 Setpoint Maximum" %
%   N17:0  TIC111_CNTL  "TIC-11-1 Tempered Water No-1 Control Word" %
%   N17:24  TIC111_IN  "TIC-11-1 Tempered Water No-1 Scaled Input" %
%   N18:21  TIC111_OUT1  "TIC-11-1 Tempered Water No-1 PID Output Value" %

